{attribute 'linkalways'} 
{attribute 'no_explicit_call' := 'This FB is a CLASS and must be accessed using methods or properties'}
{attribute 'enable_dynamic_creation'}
FUNCTION_BLOCK FINAL SUB_LINT EXTENDS Node
VAR
	in1 : _LINT(0);
	in2 : _LINT(0);
	out : _LINT(0);
END_VAR

METHOD PUBLIC Clone : I_Node
VAR
	pNode : POINTER TO SUB_LINT;
END_VAR
pNode := __NEW(SUB_LINT);
Clone := pNode^;
END_METHOD

METHOD FB_init : BOOL
VAR_INPUT
	bInitRetains : BOOL; // if TRUE, the retain variables are initialized (warm start / cold start)
	bInCopyCode : BOOL;  // if TRUE, the instance afterwards gets moved into the copy code (online change)
END_VAR
AddInput('in1',THIS^.in1);
AddInput('in2',THIS^.in2);
AddOutput('out', THIS^.out);
END_METHOD

METHOD PROTECTED OnExecute
VAR
END_VAR
out.Value := in1.Value - in2.Value;
END_METHOD

END_FUNCTION_BLOCK

(* stored: Version 1.1.0.1, ProductVersion 3.1.4024.15
   POU SUB_LINT: Id {0dc0d494-cbcb-4f9f-b2a9-e115c5c64559}, SpecialFunc None
   Folder Constructor: Id {760f4f4a-6c04-4602-b008-f97c45ef8d6b}
   Method Clone: Id {d9a4706b-143b-4d7a-a8da-8fc0a2554ac3}
   Method FB_init: Id {509e8bae-1c5e-457a-8eb8-d2747d475e46}
   Method OnExecute: Id {1f049a55-f411-4274-8d03-530c3ce4c9b1} *)
